LIN {X 0,Y 113.358,Z 438.238,A -85,B 0,C 180,E1 -30047.539,E2 -30047.539} C_VEL
LIN {X 0,Y 106.074,Z 444.931,A -85,B 0,C 180,E1 -30048.777,E2 -30048.777} C_VEL
LIN {X 0,Y 99.927,Z 449.702,A -85,B 0,C 180,E1 -30049.935,E2 -30049.935} C_VEL
LIN {X 0,Y 90.469,Z 455.663,A -85,B 0,C 180,E1 -30052.07,E2 -30052.07} C_VEL
LIN {X 0,Y 80.28,Z 460.656,A -85,B 0,C 180,E1 -30054.978,E2 -30054.978} C_VEL
LIN {X 0,Y 70.292,Z 464.167,A -85,B 0,C 180,E1 -30058.832,E2 -30058.832} C_VEL
LIN {X 0,Y 63.307,Z 465.896,A -85,B 0,C 180,E1 -30062.433,E2 -30062.433} C_VEL
LIN {X 0,Y 56.331,Z 466.986,A -85,B 0,C 180,E1 -30067.168,E2 -30067.168} C_VEL
LIN {X 0,Y 50.39,Z 467.331,A -85,B 0,C 180,E1 -30072.508,E2 -30072.508} C_VEL
LIN {X 0,Y 44.748,Z 467.097,A -85,B 0,C 180,E1 -30079.556,E2 -30079.556} C_VEL
LIN {X 0,Y 38.027,Z 465.658,A -85,B 0,C 180,E1 -30093.674,E2 -30093.674} C_VEL
LIN {X 0,Y 34.275,Z 462.616,A -85,B 0,C 180,E1 -30112.04,E2 -30112.04} C_VEL
LIN {X 0,Y 33.895,Z 459.781,A -85,B 0,C 180,E1 -30125.501,E2 -30125.501} C_VEL
LIN {X 0,Y 35.6,Z 455.392,A -85,B 0,C 180,E1 -30140.788,E2 -30140.788} C_VEL
LIN {X 0,Y 38.607,Z 450.53,A -85,B 0,C 180,E1 -30152.609,E2 -30152.609} C_VEL
LIN {X 0,Y 42.581,Z 444.846,A -85,B 0,C 180,E1 -30162.061,E2 -30162.061} C_VEL
LIN {X 0,Y 46.328,Z 439.524,A -85,B 0,C 180,E1 -30168.255,E2 -30168.255} C_VEL
LIN {X 0,Y 48.568,Z 435.44,A -85,B 0,C 180,E1 -30172.498,E2 -30172.498} C_VEL
LIN {X 0,Y 51.052,Z 428.248,A -85,B 0,C 180,E1 -30179.49,E2 -30179.49} C_VEL
LIN {X 0,Y 53.719,Z 420.249,A -85,B 0,C 180,E1 -30185.421,E2 -30185.421} C_VEL
LIN {X 0,Y 55.987,Z 414.967,A -85,B 0,C 180,E1 -30187.677,E2 -30187.677} C_VEL
LIN {X 0,Y 60.515,Z 403.977,A -85,B 0,C 180,E1 -30190.224,E2 -30190.224} C_VEL
LIN {X 0,Y 63.497,Z 393.798,A -85,B 0,C 180,E1 -30191.853,E2 -30191.853} C_VEL
LIN {X 0,Y 65.38,Z 384.895,A -85,B 0,C 180,E1 -30192.729,E2 -30192.729} C_VEL
LIN {X 0,Y 66.668,Z 375.67,A -85,B 0,C 180,E1 -30193.366,E2 -30193.366} C_VEL
LIN {X 0,Y 64.802,Z 370.412,A -85,B 0,C 180,E1 -30197.601,E2 -30197.601} C_VEL
LIN {X 0,Y 62.957,Z 365.838,A -85,B 0,C 180,E1 -30202.626,E2 -30202.626} C_VEL
LIN {X 0,Y 61.544,Z 362.657,A -85,B 0,C 180,E1 -30207.536,E2 -30207.536} C_VEL
LIN {X 0,Y 60.692,Z 360.754,A -85,B 0,C 180,E1 -30211.237,E2 -30211.237} C_VEL
LIN {X 0,Y 59.513,Z 357.859,A -85,B 0,C 180,E1 -30220.097,E2 -30220.097} C_VEL
LIN {X 0,Y 59.44,Z 356.985,A -85,B 0,C 180,E1 -30222.889,E2 -30222.889} C_VEL
LIN {X 0,Y 59.712,Z 357.064,A -85,B 0,C 180,E1 -30232.39,E2 -30232.39} C_VEL
LIN {X 0,Y 60.992,Z 360.897,A -85,B 0,C 180,E1 -30241.472,E2 -30241.472} C_VEL
LIN {X 0,Y 62.477,Z 364.593,A -85,B 0,C 180,E1 -30247.411,E2 -30247.411} C_VEL
LIN {X 0,Y 64.572,Z 369.926,A -85,B 0,C 180,E1 -30253.445,E2 -30253.445} C_VEL
LIN {X 0,Y 66.7,Z 376.361,A -85,B 0,C 180,E1 -30258.427,E2 -30258.427} C_VEL
LIN {X 0,Y 64.594,Z 390.953,A -85,B 0,C 180,E1 -30259.542,E2 -30259.542} C_VEL
LIN {X 0,Y 61.713,Z 401.445,A -85,B 0,C 180,E1 -30260.693,E2 -30260.693} C_VEL
LIN {X 0,Y 58.801,Z 409.625,A -85,B 0,C 180,E1 -30262.14,E2 -30262.14} C_VEL
LIN {X 0,Y 54.998,Z 418.265,A -85,B 0,C 180,E1 -30264.433,E2 -30264.433} C_VEL
LIN {X 0,Y 50.429,Z 426.455,A -85,B 0,C 180,E1 -30267.325,E2 -30267.325} C_VEL
LIN {X 0,Y 45.461,Z 434.326,A -85,B 0,C 180,E1 -30271.761,E2 -30271.761} C_VEL
LIN {X 0,Y 40.078,Z 441.645,A -85,B 0,C 180,E1 -30277.899,E2 -30277.899} C_VEL
LIN {X 0,Y 34.266,Z 449.088,A -85,B 0,C 180,E1 -30288.197,E2 -30288.197} C_VEL
LIN {X 0,Y 29.923,Z 454.906,A -85,B 0,C 180,E1 -30301.984,E2 -30301.984} C_VEL
LIN {X 0,Y 27.869,Z 458.679,A -85,B 0,C 180,E1 -30315.394,E2 -30315.394} C_VEL
LIN {X 0,Y 27.402,Z 461.71,A -85,B 0,C 180,E1 -30330,E2 -30330} C_VEL
LIN {X 0,Y 27.953,Z 464.041,A -85,B 0,C 180,E1 -30344.561,E2 -30344.561} C_VEL
LIN {X 0,Y 29.91,Z 465.846,A -85,B 0,C 180,E1 -30358.029,E2 -30358.029} C_VEL
LIN {X 0,Y 33.278,Z 467.197,A -85,B 0,C 180,E1 -30369.312,E2 -30369.312} C_VEL
LIN {X 0,Y 37.711,Z 468.061,A -85,B 0,C 180,E1 -30378.196,E2 -30378.196} C_VEL
LIN {X 0,Y 42.805,Z 468.367,A -85,B 0,C 180,E1 -30385.174,E2 -30385.174} C_VEL
LIN {X 0,Y 48.486,Z 468.264,A -85,B 0,C 180,E1 -30390.42,E2 -30390.42} C_VEL
LIN {X 0,Y 54.509,Z 467.751,A -85,B 0,C 180,E1 -30394.489,E2 -30394.489} C_VEL
LIN {X 0,Y 60.791,Z 466.752,A -85,B 0,C 180,E1 -30397.644,E2 -30397.644} C_VEL
LIN {X 0,Y 70.486,Z 464.294,A -85,B 0,C 180,E1 -30401.296,E2 -30401.296} C_VEL
LIN {X 0,Y 80.377,Z 460.617,A -85,B 0,C 180,E1 -30404.11,E2 -30404.11} C_VEL
LIN {X 0,Y 87.09,Z 457.513,A -85,B 0,C 180,E1 -30405.545,E2 -30405.545} C_VEL
LIN {X 0,Y 93.853,Z 453.722,A -85,B 0,C 180,E1 -30406.768,E2 -30406.768} C_VEL
LIN {X 0,Y 86.139,Z 457.911,A -85,B 0,C 180,E1 -30408.248,E2 -30408.248} C_VEL
LIN {X 0,Y 78.492,Z 461.253,A -85,B 0,C 180,E1 -30410.026,E2 -30410.026} C_VEL
LIN {X 0,Y 70.931,Z 463.82,A -85,B 0,C 180,E1 -30412.215,E2 -30412.215} C_VEL
LIN {X 0,Y 63.486,Z 465.68,A -85,B 0,C 180,E1 -30415.059,E2 -30415.059} C_VEL
LIN {X 0,Y 53.864,Z 467.215,A -85,B 0,C 180,E1 -30420.001,E2 -30420.001} C_VEL
LIN {X 0,Y 42.371,Z 467.398,A -85,B 0,C 180,E1 -30429.549,E2 -30429.549} C_VEL
LIN {X 0,Y 36.786,Z 466.766,A -85,B 0,C 180,E1 -30437.214,E2 -30437.214} C_VEL
LIN {X 0,Y 31.83,Z 465.482,A -85,B 0,C 180,E1 -30447.974,E2 -30447.974} C_VEL
LIN {X 0,Y 28.313,Z 463.542,A -85,B 0,C 180,E1 -30461.872,E2 -30461.872} C_VEL
LIN {X 0,Y 26.781,Z 460.888,A -85,B 0,C 180,E1 -30478.343,E2 -30478.343} C_VEL
LIN {X 0,Y 27.49,Z 457.48,A -85,B 0,C 180,E1 -30495.188,E2 -30495.188} C_VEL
LIN {X 0,Y 30.877,Z 452.116,A -85,B 0,C 180,E1 -30513.262,E2 -30513.262} C_VEL
LIN {X 0,Y 35.633,Z 446.024,A -85,B 0,C 180,E1 -30525.772,E2 -30525.772} C_VEL
LIN {X 0,Y 40.971,Z 439.218,A -85,B 0,C 180,E1 -30534.372,E2 -30534.372} C_VEL
LIN {X 0,Y 45.827,Z 432.472,A -85,B 0,C 180,E1 -30539.895,E2 -30539.895} C_VEL
LIN {X 0,Y 50.437,Z 425.276,A -85,B 0,C 180,E1 -30543.873,E2 -30543.873} C_VEL
LIN {X 0,Y 54.378,Z 418.101,A -85,B 0,C 180,E1 -30546.711,E2 -30546.711} C_VEL
LIN {X 0,Y 55.987,Z 414.967,A -85,B 0,C 180,E1 -30547.677,E2 -30547.677} C_VEL
LIN {X 0,Y 57.249,Z 411.509,A -85,B 0,C 180,E1 -30549.246,E2 -30549.246} C_VEL
LIN {X 0,Y 58.01,Z 405.904,A -85,B 0,C 180,E1 -30552.97,E2 -30552.97} C_VEL
LIN {X 0,Y 58.575,Z 400.09,A -85,B 0,C 180,E1 -30556.356,E2 -30556.356} C_VEL
LIN {X 0,Y 59.363,Z 396.303,A -85,B 0,C 180,E1 -30557.319,E2 -30557.319} C_VEL
LIN {X 0,Y 61.827,Z 385.703,A -85,B 0,C 180,E1 -30558.248,E2 -30558.248} C_VEL
LIN {X 0,Y 62.962,Z 378.303,A -85,B 0,C 180,E1 -30558.752,E2 -30558.752} C_VEL
LIN {X 0,Y 61.458,Z 373.492,A -85,B 0,C 180,E1 -30563.497,E2 -30563.497} C_VEL
LIN {X 0,Y 60.009,Z 369.419,A -85,B 0,C 180,E1 -30569.299,E2 -30569.299} C_VEL
LIN {X 0,Y 59.254,Z 367.413,A -85,B 0,C 180,E1 -30573.294,E2 -30573.294} C_VEL
LIN {X 0,Y 58.438,Z 364.244,A -85,B 0,C 180,E1 -30582.985,E2 -30582.985} C_VEL
LIN {X 0,Y 58.418,Z 363.941,A -85,B 0,C 180,E1 -30586.077,E2 -30586.077} C_VEL
LIN {X 0,Y 58.604,Z 364.053,A -85,B 0,C 180,E1 -30590.943,E2 -30590.943} C_VEL
LIN {X 0,Y 59.4,Z 367.232,A -85,B 0,C 180,E1 -30598.804,E2 -30598.804} C_VEL
LIN {X 0,Y 60.792,Z 371.447,A -85,B 0,C 180,E1 -30605.604,E2 -30605.604} C_VEL
LIN {X 0,Y 62.287,Z 376.327,A -85,B 0,C 180,E1 -30610.916,E2 -30610.916} C_VEL
LIN {X 0,Y 63.005,Z 378.972,A -85,B 0,C 180,E1 -30613.114,E2 -30613.114} C_VEL
LIN {X 0,Y 60.767,Z 392.16,A -85,B 0,C 180,E1 -30614.059,E2 -30614.059} C_VEL
LIN {X 0,Y 57.735,Z 402.294,A -85,B 0,C 180,E1 -30614.965,E2 -30614.965} C_VEL
LIN {X 0,Y 54.069,Z 411.701,A -85,B 0,C 180,E1 -30616.548,E2 -30616.548} C_VEL
LIN {X 0,Y 50.03,Z 419.865,A -85,B 0,C 180,E1 -30618.525,E2 -30618.525} C_VEL
LIN {X 0,Y 44.451,Z 428.984,A -85,B 0,C 180,E1 -30621.745,E2 -30621.745} C_VEL
LIN {X 0,Y 37.616,Z 438.228,A -85,B 0,C 180,E1 -30627.445,E2 -30627.445} C_VEL
LIN {X 0,Y 31.971,Z 444.799,A -85,B 0,C 180,E1 -30634.481,E2 -30634.481} C_VEL
LIN {X 0,Y 26.957,Z 450.254,A -85,B 0,C 180,E1 -30644.197,E2 -30644.197} C_VEL
LIN {X 0,Y 22.271,Z 455.759,A -85,B 0,C 180,E1 -30661.748,E2 -30661.748} C_VEL
LIN {X 0,Y 20.349,Z 460.839,A -85,B 0,C 180,E1 -30690,E2 -30690} C_VEL
LIN {X 0,Y 21.183,Z 463.331,A -85,B 0,C 180,E1 -30709.375,E2 -30709.375} C_VEL
LIN {X 0,Y 23.896,Z 465.288,A -85,B 0,C 180,E1 -30726.029,E2 -30726.029} C_VEL
LIN {X 0,Y 28.151,Z 466.752,A -85,B 0,C 180,E1 -30738.498,E2 -30738.498} C_VEL
LIN {X 0,Y 33.404,Z 467.644,A -85,B 0,C 180,E1 -30747.302,E2 -30747.302} C_VEL
LIN {X 0,Y 39.181,Z 468.093,A -85,B 0,C 180,E1 -30753.745,E2 -30753.745} C_VEL
LIN {X 0,Y 45.407,Z 468.145,A -85,B 0,C 180,E1 -30758.223,E2 -30758.223} C_VEL
LIN {X 0,Y 51.852,Z 467.752,A -85,B 0,C 180,E1 -30761.576,E2 -30761.576} C_VEL
LIN {X 0,Y 58.458,Z 466.791,A -85,B 0,C 180,E1 -30764.101,E2 -30764.101} C_VEL
LIN {X 0,Y 65.154,Z 465.377,A -85,B 0,C 180,E1 -30766.115,E2 -30766.115} C_VEL
LIN {X 0,Y 65.485,Z 465.254,A -85,B 0,C 180,E1 -30767.606,E2 -30767.606} C_VEL
LIN {X 0,Y 52.336,Z 467.443,A -85,B 0,C 180,E1 -30772.284,E2 -30772.284} C_VEL
LIN {X 0,Y 39.763,Z 467.597,A -85,B 0,C 180,E1 -30780.001,E2 -30780.001} C_VEL
LIN {X 0,Y 35.241,Z 467.267,A -85,B 0,C 180,E1 -30784.361,E2 -30784.361} C_VEL
LIN {X 0,Y 28.528,Z 466.032,A -85,B 0,C 180,E1 -30794.263,E2 -30794.263} C_VEL
LIN {X 0,Y 21.864,Z 463.271,A -85,B 0,C 180,E1 -30815.044,E2 -30815.044} C_VEL
LIN {X 0,Y 19.717,Z 460.347,A -85,B 0,C 180,E1 -30837.681,E2 -30837.681} C_VEL
LIN {X 0,Y 21.199,Z 455.982,A -85,B 0,C 180,E1 -30864.062,E2 -30864.062} C_VEL
LIN {X 0,Y 25.218,Z 451.124,A -85,B 0,C 180,E1 -30882.064,E2 -30882.064} C_VEL
LIN {X 0,Y 31.064,Z 444.775,A -85,B 0,C 180,E1 -30895.179,E2 -30895.179} C_VEL
LIN {X 0,Y 36.239,Z 438.857,A -85,B 0,C 180,E1 -30902.229,E2 -30902.229} C_VEL
LIN {X 0,Y 42.647,Z 430.626,A -85,B 0,C 180,E1 -30908.167,E2 -30908.167} C_VEL
LIN {X 0,Y 49.006,Z 420.737,A -85,B 0,C 180,E1 -30912.407,E2 -30912.407} C_VEL
LIN {X 0,Y 53.556,Z 411.907,A -85,B 0,C 180,E1 -30914.714,E2 -30914.714} C_VEL
LIN {X 0,Y 57.439,Z 402.293,A -85,B 0,C 180,E1 -30916.431,E2 -30916.431} C_VEL
LIN {X 0,Y 59.363,Z 396.303,A -85,B 0,C 180,E1 -30917.319,E2 -30917.319} C_VEL
LIN {X 0,Y 60.206,Z 392.362,A -85,B 0,C 180,E1 -30918.064,E2 -30918.064} C_VEL
LIN {X 0,Y 60.549,Z 388.565,A -85,B 0,C 180,E1 -30919.583,E2 -30919.583} C_VEL
LIN {X 0,Y 60.248,Z 383.907,A -85,B 0,C 180,E1 -30922.417,E2 -30922.417} C_VEL
LIN {X 0,Y 59.549,Z 379.893,A -85,B 0,C 180,E1 -30926.084,E2 -30926.084} C_VEL
LIN {X 0,Y 59.091,Z 378.204,A -85,B 0,C 180,E1 -30928.197,E2 -30928.197} C_VEL
LIN {X 0,Y 57.989,Z 374.198,A -85,B 0,C 180,E1 -30934.843,E2 -30934.843} C_VEL
LIN {X 0,Y 57.459,Z 371.029,A -85,B 0,C 180,E1 -30944.871,E2 -30944.871} C_VEL
LIN {X 0,Y 57.539,Z 371.132,A -85,B 0,C 180,E1 -30949.72,E2 -30949.72} C_VEL
LIN {X 0,Y 58.006,Z 373.961,A -85,B 0,C 180,E1 -30956.655,E2 -30956.655} C_VEL
LIN {X 0,Y 58.918,Z 377.52,A -85,B 0,C 180,E1 -30962.481,E2 -30962.481} C_VEL
LIN {X 0,Y 59.835,Z 381.563,A -85,B 0,C 180,E1 -30967.014,E2 -30967.014} C_VEL
LIN {X 0,Y 57.709,Z 392.756,A -85,B 0,C 180,E1 -30967.847,E2 -30967.847} C_VEL
LIN {X 0,Y 54.993,Z 401.577,A -85,B 0,C 180,E1 -30968.345,E2 -30968.345} C_VEL
LIN {X 0,Y 51.427,Z 410.542,A -85,B 0,C 180,E1 -30969.449,E2 -30969.449} C_VEL
LIN {X 0,Y 47.406,Z 418.519,A -85,B 0,C 180,E1 -30970.849,E2 -30970.849} C_VEL
LIN {X 0,Y 42.335,Z 426.604,A -85,B 0,C 180,E1 -30972.767,E2 -30972.767} C_VEL
LIN {X 0,Y 37.392,Z 433.367,A -85,B 0,C 180,E1 -30975.582,E2 -30975.582} C_VEL
LIN {X 0,Y 31.702,Z 439.923,A -85,B 0,C 180,E1 -30979.583,E2 -30979.583} C_VEL
LIN {X 0,Y 25.514,Z 446.176,A -85,B 0,C 180,E1 -30986.464,E2 -30986.464} C_VEL
LIN {X 0,Y 19.895,Z 451.354,A -85,B 0,C 180,E1 -30997.362,E2 -30997.362} C_VEL
LIN {X 0,Y 14.615,Z 456.595,A -85,B 0,C 180,E1 -31021.258,E2 -31021.258} C_VEL
LIN {X 0,Y 13.271,Z 459.946,A -85,B 0,C 180,E1 -31049.999,E2 -31049.999} C_VEL
LIN {X 0,Y 14.708,Z 462.598,A -85,B 0,C 180,E1 -31078.542,E2 -31078.542} C_VEL
LIN {X 0,Y 18.647,Z 464.695,A -85,B 0,C 180,E1 -31098.917,E2 -31098.917} C_VEL
LIN {X 0,Y 24.048,Z 466.194,A -85,B 0,C 180,E1 -31111.248,E2 -31111.248} C_VEL
LIN {X 0,Y 30.163,Z 467.216,A -85,B 0,C 180,E1 -31118.744,E2 -31118.744} C_VEL
LIN {X 0,Y 36.595,Z 467.82,A -85,B 0,C 180,E1 -31123.78,E2 -31123.78} C_VEL
LIN {X 0,Y 43.238,Z 468.012,A -85,B 0,C 180,E1 -31127.218,E2 -31127.218} C_VEL
LIN {X 0,Y 35.566,Z 467.637,A -85,B 0,C 180,E1 -31131.108,E2 -31131.108} C_VEL
LIN {X 0,Y 25.644,Z 466.205,A -85,B 0,C 180,E1 -31140.002,E2 -31140.002} C_VEL
LIN {X 0,Y 18.173,Z 464.023,A -85,B 0,C 180,E1 -31154.807,E2 -31154.807} C_VEL
LIN {X 0,Y 13.419,Z 461.228,A -85,B 0,C 180,E1 -31180.855,E2 -31180.855} C_VEL
LIN {X 0,Y 14.063,Z 456.216,A -85,B 0,C 180,E1 -31228.329,E2 -31228.329} C_VEL
LIN {X 0,Y 19.047,Z 451.383,A -85,B 0,C 180,E1 -31251.653,E2 -31251.653} C_VEL
LIN {X 0,Y 25.773,Z 445.196,A -85,B 0,C 180,E1 -31265.106,E2 -31265.106} C_VEL
LIN {X 0,Y 31.736,Z 439.169,A -85,B 0,C 180,E1 -31271.632,E2 -31271.632} C_VEL
LIN {X 0,Y 37.833,Z 432.067,A -85,B 0,C 180,E1 -31276.039,E2 -31276.039} C_VEL
LIN {X 0,Y 44.786,Z 422.32,A -85,B 0,C 180,E1 -31279.594,E2 -31279.594} C_VEL
LIN {X 0,Y 50.364,Z 412.157,A -85,B 0,C 180,E1 -31281.712,E2 -31281.712} C_VEL
LIN {X 0,Y 54.307,Z 402.874,A -85,B 0,C 180,E1 -31282.972,E2 -31282.972} C_VEL
LIN {X 0,Y 57.233,Z 393.565,A -85,B 0,C 180,E1 -31283.961,E2 -31283.961} C_VEL
LIN {X 0,Y 59.289,Z 384.334,A -85,B 0,C 180,E1 -31284.507,E2 -31284.507} C_VEL
LIN {X 0,Y 59.796,Z 381.147,A -85,B 0,C 180,E1 -31284.808,E2 -31284.808} C_VEL
LIN {X 0,Y 59.091,Z 378.204,A -85,B 0,C 180,E1 -31288.197,E2 -31288.197} C_VEL
LIN {X 0,Y 58.345,Z 376.562,A -85,B 0,C 180,E1 -31291.681,E2 -31291.681} C_VEL
LIN {X 0,Y 57.411,Z 375.915,A -85,B 0,C 180,E1 -31296.896,E2 -31296.896} C_VEL
LIN {X 0,Y 56.676,Z 376.865,A -85,B 0,C 180,E1 -31303.805,E2 -31303.805} C_VEL
LIN {X 0,Y 56.502,Z 378.487,A -85,B 0,C 180,E1 -31309.278,E2 -31309.278} C_VEL
LIN {X 0,Y 56.666,Z 380.38,A -85,B 0,C 180,E1 -31313.858,E2 -31313.858} C_VEL
LIN {X 0,Y 57.063,Z 383.354,A -85,B 0,C 180,E1 -31318.897,E2 -31318.897} C_VEL
LIN {X 0,Y 57.223,Z 384.656,A -85,B 0,C 180,E1 -31320.575,E2 -31320.575} C_VEL
LIN {X 0,Y 55.338,Z 393.412,A -85,B 0,C 180,E1 -31321.01,E2 -31321.01} C_VEL
LIN {X 0,Y 52.178,Z 403.073,A -85,B 0,C 180,E1 -31321.226,E2 -31321.226} C_VEL
LIN {X 0,Y 48.344,Z 412.036,A -85,B 0,C 180,E1 -31321.954,E2 -31321.954} C_VEL
LIN {X 0,Y 43.972,Z 420.014,A -85,B 0,C 180,E1 -31322.692,E2 -31322.692} C_VEL
LIN {X 0,Y 37.872,Z 429.049,A -85,B 0,C 180,E1 -31324.121,E2 -31324.121} C_VEL
LIN {X 0,Y 30.077,Z 438.127,A -85,B 0,C 180,E1 -31326.757,E2 -31326.757} C_VEL
LIN {X 0,Y 23.239,Z 444.635,A -85,B 0,C 180,E1 -31330.629,E2 -31330.629} C_VEL
LIN {X 0,Y 16.577,Z 450.039,A -85,B 0,C 180,E1 -31337.465,E2 -31337.465} C_VEL
LIN {X 0,Y 9.08,Z 455.491,A -85,B 0,C 180,E1 -31359.287,E2 -31359.287} C_VEL
LIN {X 0,Y 6.206,Z 459.029,A -85,B 0,C 180,E1 -31409.999,E2 -31409.999} C_VEL
LIN {X 0,Y 9.151,Z 461.85,A -85,B 0,C 180,E1 -31460.17,E2 -31460.17} C_VEL
LIN {X 0,Y 14.982,Z 464.001,A -85,B 0,C 180,E1 -31479.743,E2 -31479.743} C_VEL
LIN {X 0,Y 17.554,Z 464.673,A -85,B 0,C 180,E1 -31488.998,E2 -31488.998} C_VEL
LIN {X 0,Y 7.429,Z 460.829,A -85,B 0,C 180,E1 -31518.926,E2 -31518.926} C_VEL
LIN {X 0,Y 7.173,Z 456.405,A -85,B 0,C 180,E1 -31601.491,E2 -31601.491} C_VEL
LIN {X 0,Y 13.863,Z 451.613,A -85,B 0,C 180,E1 -31629.324,E2 -31629.324} C_VEL
LIN {X 0,Y 21.546,Z 445.637,A -85,B 0,C 180,E1 -31639.276,E2 -31639.276} C_VEL
LIN {X 0,Y 28.365,Z 439.389,A -85,B 0,C 180,E1 -31643.633,E2 -31643.633} C_VEL
LIN {X 0,Y 35.491,Z 431.544,A -85,B 0,C 180,E1 -31646.481,E2 -31646.481} C_VEL
LIN {X 0,Y 42.306,Z 422.309,A -85,B 0,C 180,E1 -31648.36,E2 -31648.36} C_VEL
LIN {X 0,Y 47.913,Z 412.439,A -85,B 0,C 180,E1 -31649.512,E2 -31649.512} C_VEL
LIN {X 0,Y 52.195,Z 402.611,A -85,B 0,C 180,E1 -31650.247,E2 -31650.247} C_VEL
LIN {X 0,Y 55.185,Z 393.274,A -85,B 0,C 180,E1 -31650.875,E2 -31650.875} C_VEL
LIN {X 0,Y 57.151,Z 384.584,A -85,B 0,C 180,E1 -31651.179,E2 -31651.179} C_VEL
LIN {X 0,Y 56.752,Z 381.539,A -85,B 0,C 180,E1 -31655.875,E2 -31655.875} C_VEL
LIN {X 0,Y 56.501,Z 380.267,A -85,B 0,C 180,E1 -31659.296,E2 -31659.296} C_VEL
LIN {X 0,Y 56.49,Z 377.99,A -85,B 0,C 180,E1 -31666.682,E2 -31666.682} C_VEL
LIN {X 0,Y 56.501,Z 378.341,A -85,B 0,C 180,E1 -31668.858,E2 -31668.858} C_VEL
LIN {X 0,Y 56.502,Z 378.487,A -85,B 0,C 180,E1 -31669.278,E2 -31669.278} C_VEL
LIN {X 0,Y 56.458,Z 379.891,A -85,B 0,C 180,E1 -31671.373,E2 -31671.373} C_VEL
LIN {X 0,Y 56.219,Z 382.596,A -85,B 0,C 180,E1 -31673.121,E2 -31673.121} C_VEL
LIN {X 0,Y 55.516,Z 387.094,A -85,B 0,C 180,E1 -31674.199,E2 -31674.199} C_VEL
LIN {X 0,Y 54.103,Z 393.082,A -85,B 0,C 180,E1 -31674.048,E2 -31674.048} C_VEL
LIN {X 0,Y 52.296,Z 398.969,A -85,B 0,C 180,E1 -31673.559,E2 -31673.559} C_VEL
LIN {X 0,Y 48.394,Z 408.797,A -85,B 0,C 180,E1 -31673.497,E2 -31673.497} C_VEL
LIN {X 0,Y 44.201,Z 417.031,A -85,B 0,C 180,E1 -31673.58,E2 -31673.58} C_VEL
LIN {X 0,Y 38.916,Z 425.292,A -85,B 0,C 180,E1 -31673.337,E2 -31673.337} C_VEL
LIN {X 0,Y 32.72,Z 433.209,A -85,B 0,C 180,E1 -31673.411,E2 -31673.411} C_VEL
LIN {X 0,Y 26.542,Z 439.718,A -85,B 0,C 180,E1 -31673.173,E2 -31673.173} C_VEL
LIN {X 0,Y 19.964,Z 445.53,A -85,B 0,C 180,E1 -31672.761,E2 -31672.761} C_VEL
LIN {X 0,Y 12.424,Z 451.066,A -85,B 0,C 180,E1 -31671.853,E2 -31671.853} C_VEL
LIN {X 0,Y 7.149,Z 454.389,A -85,B 0,C 180,E1 -31669.448,E2 -31669.448} C_VEL
LIN {X 0,Y 7.302,Z 454.284,A -85,B 0,C 180,E1 -31664.251,E2 -31664.251} C_VEL
LIN {X 0,Y 17.479,Z 447.443,A -85,B 0,C 180,E1 -31658.781,E2 -31658.781} C_VEL
LIN {X 0,Y 24.609,Z 441.458,A -85,B 0,C 180,E1 -31658.145,E2 -31658.145} C_VEL
LIN {X 0,Y 32.199,Z 433.635,A -85,B 0,C 180,E1 -31658.076,E2 -31658.076} C_VEL
LIN {X 0,Y 37.905,Z 426.514,A -85,B 0,C 180,E1 -31657.976,E2 -31657.976} C_VEL
LIN {X 0,Y 42.644,Z 419.426,A -85,B 0,C 180,E1 -31657.975,E2 -31657.975} C_VEL
LIN {X 0,Y 47.516,Z 410.427,A -85,B 0,C 180,E1 -31657.945,E2 -31657.945} C_VEL
LIN {X 0,Y 51.202,Z 401.689,A -85,B 0,C 180,E1 -31658.033,E2 -31658.033} C_VEL
LIN {X 0,Y 54.324,Z 391.68,A -85,B 0,C 180,E1 -31658.209,E2 -31658.209} C_VEL
LIN {X 0,Y 55.206,Z 388.123,A -85,B 0,C 180,E1 -31658.213,E2 -31658.213} C_VEL
LIN {X 0,Y 55.134,Z 386.848,A -85,B 0,C 180,E1 -31661.615,E2 -31661.615} C_VEL
LIN {X 0,Y 55.304,Z 385.331,A -85,B 0,C 180,E1 -31667.509,E2 -31667.509} C_VEL
LIN {X 0,Y 55.22,Z 387.26,A -85,B 0,C 180,E1 -31671.944,E2 -31671.944} C_VEL
LIN {X 0,Y 55.249,Z 388.065,A -85,B 0,C 180,E1 -31673.528,E2 -31673.528} C_VEL
LIN {X 0,Y 53.379,Z 395.38,A -85,B 0,C 180,E1 -31673.648,E2 -31673.648} C_VEL
LIN {X 0,Y 52.296,Z 398.969,A -85,B 0,C 180,E1 -31673.559,E2 -31673.559} C_VEL
LIN {X 0,Y 52.188,Z 399.617,A -85,B 0,C 180,E1 -31673.546,E2 -31673.546} C_VEL
LIN {X 0,Y 52.188,Z 600,A -85,B 0,C 180,E1 -31673.546,E2 -31673.546} C_VEL
LIN {X 0,Y 52.188,Z 600,A -85,B 0,C 180,E1 -31673.546,E2 -31673.546}

QRS_NEXT_CUT()

QRS_NEXT()
QRS_HOME()

END
